// TIA Portal project "BatchSimulation_S71500" (V15)

(* hardware
DEVICE "S71500/ET200MP station_1"  S7-1500 station
   slot 0: "Rail_0"  Rack  6ES7 590-1***0-0AA0
   slot 1: "PLC_2_BatchController"  CPU 1512C-1 PN  6ES7 512-1CK01-0AB0  V2.5
      slot 3: "CPU display_1"  6ES7591-1AA00-0AA0
DEVICE "S71500/ET200MP station_2"  S7-1500 station
   slot 0: "Rail_0"  Rack  6ES7 590-1***0-0AA0
   slot 1: "PLC_1_Master"  CPU 1512C-1 PN  6ES7 512-1CK01-0AB0  V2.5
      slot 3: "CPU display_1"  6ES7591-1AA00-0AA0
*)

// ===== PLC "PLC_2_BatchController"  CPU 1512C-1 PN =====

VAR_GLOBAL   // PLC tag table "Default tag table"
   "Enable" AT %M100.0 : Bool;
   "Start" AT %M100.1 : Bool;
   "Estop" AT %M100.2 : Bool;
   "Ready" AT %M100.3 : Bool;
   "Setpoint" AT %MD150 : Real;
   "Vout" AT %MD154 : Real;
   "Running" AT %M100.4 : Bool;
   "State" AT %MW200 : Int;
   "Tag_1" AT %MD1000 : Real;
   "Tag_2" AT %MD1004 : DWord;
   "Tag_3" AT %M50.0 : Bool;
   "Tag_4" AT %M200.0 : Bool;
   "Tag_5" AT %MW204 : Int;
   "Tag_6" AT %M700.0 : Bool;
   "Tag_7" AT %MD200 : Real;
   "Tag_8" AT %MD300 : Real;
   "Tag_9" AT %M11.0 : Bool;
   "Tag_10" AT %M10.0 : Bool;
   "System_Byte" AT %MB1 : Byte;
   "FirstScan" AT %M1.0 : Bool;
   "DiagStatusUpdate" AT %M1.1 : Bool;
   "AlwaysTRUE" AT %M1.2 : Bool;
   "AlwaysFALSE" AT %M1.3 : Bool;
END_VAR

DATA_BLOCK "Batch1_Send"   // DB4
{ S7_Optimized_Access := 'FALSE' }
VERSION : 0.1
   VAR
      Ready : Bool;
      Running : Bool;
      Clock : Bool;
      Pulse : Int := 13;
      Vout : Real;
      ctrvalue : Real;
   END_VAR
BEGIN
END_DATA_BLOCK

DATA_BLOCK "Batch1_Recv"   // DB5
{ S7_Optimized_Access := 'FALSE' }
VERSION : 0.1
   VAR
      Start : Bool;
      Estop : Bool;
      Enable : Bool;
      PS : Int;
      Setpoint : Real;
   END_VAR
BEGIN
END_DATA_BLOCK

// folder: System blocks/Program resources

DATA_BLOCK "IEC_Timer_0_DB"   // DB1
{ S7_Optimized_Access := 'TRUE' }
AUTHOR : Simatic
FAMILY : IEC
NAME : IEC_TMR
VERSION : 1.0
// stored: InstanceOfName IEC_TIMER
"IEC_TIMER"
BEGIN
END_DATA_BLOCK

DATA_BLOCK "IEC_Timer_0_DB_1"   // DB2
{ S7_Optimized_Access := 'TRUE' }
AUTHOR : Simatic
FAMILY : IEC
NAME : IEC_TMR
VERSION : 1.0
// stored: InstanceOfName IEC_TIMER
"IEC_TIMER"
BEGIN
END_DATA_BLOCK

// folder: (top level)

FUNCTION "ClockGenerator" : Void   // FC1, LAD
{ S7_Optimized_Access := 'TRUE' }
VERSION : 0.1
   VAR_INPUT
      "Flow (m3/h)" : Real;
      PS : Int;
   END_VAR
   VAR_IN_OUT
      clock : Bool;
   END_VAR
   VAR_TEMP
      timing_ms : Int;
      timing : Time;
   END_VAR
BEGIN

REGION Network 1
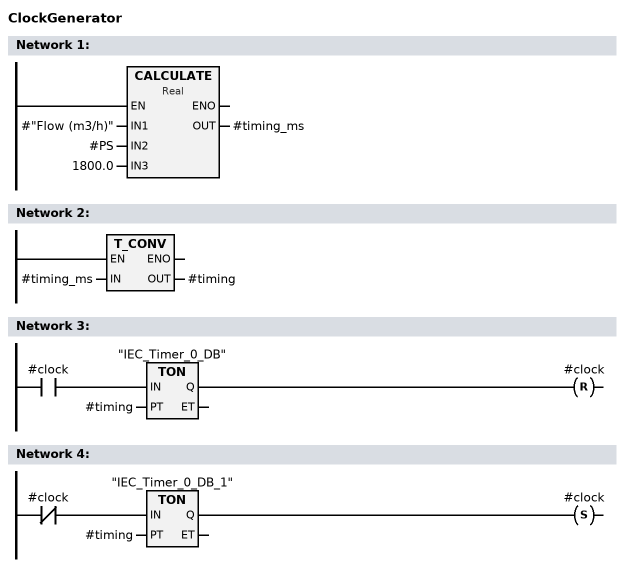
   RUNG wire#powerrail
      { S7_Templates := "SrcType := Real"; S7_Expression := "IN3/(IN1*IN2)" } Calculate(in1 := #"Flow (m3/h)", in2 := #PS, in3 := 1800.0, out => #timing_ms)
   END_RUNG
   // the same network as SCL:
   #timing_ms := 1800.0/(#"Flow (m3/h)"*#PS);
END_REGION

REGION Network 2
   #timing := T_CONV(IN := #timing_ms);
END_REGION

REGION Network 3
   "IEC_Timer_0_DB".TON(IN := #clock, PT := #timing);
   IF "IEC_Timer_0_DB".Q THEN #clock := FALSE; END_IF;
END_REGION

REGION Network 4
   "IEC_Timer_0_DB_1".TON(IN := NOT #clock, PT := #timing);
   IF "IEC_Timer_0_DB_1".Q THEN #clock := TRUE; END_IF;
END_REGION
END_FUNCTION

FUNCTION "BatchSimulation" : Void   // FC2, LAD
{ S7_Optimized_Access := 'TRUE' }
VERSION : 0.1
   VAR_INPUT
      Enable : Bool;
      Start : Bool;
      Estop : Bool;
      Setpoint : Real;
      PS : Int;
   END_VAR
   VAR_OUTPUT
      Ready : Bool;
   END_VAR
   VAR_IN_OUT
      "Vout(m3)" : Real;
      Running : Bool;
      pulse : Int;
      ctrlvalue : Real;
      clock : Bool;
   END_VAR
   VAR_TEMP
      flow : Real;
      tmp_clock : Bool;
      tmp_running : Bool;
   END_VAR
   VAR_TEMP   // added for the SCL form of the ladder/FBD networks
      _w1 : Bool;
   END_VAR
BEGIN

REGION Network 1: logic control
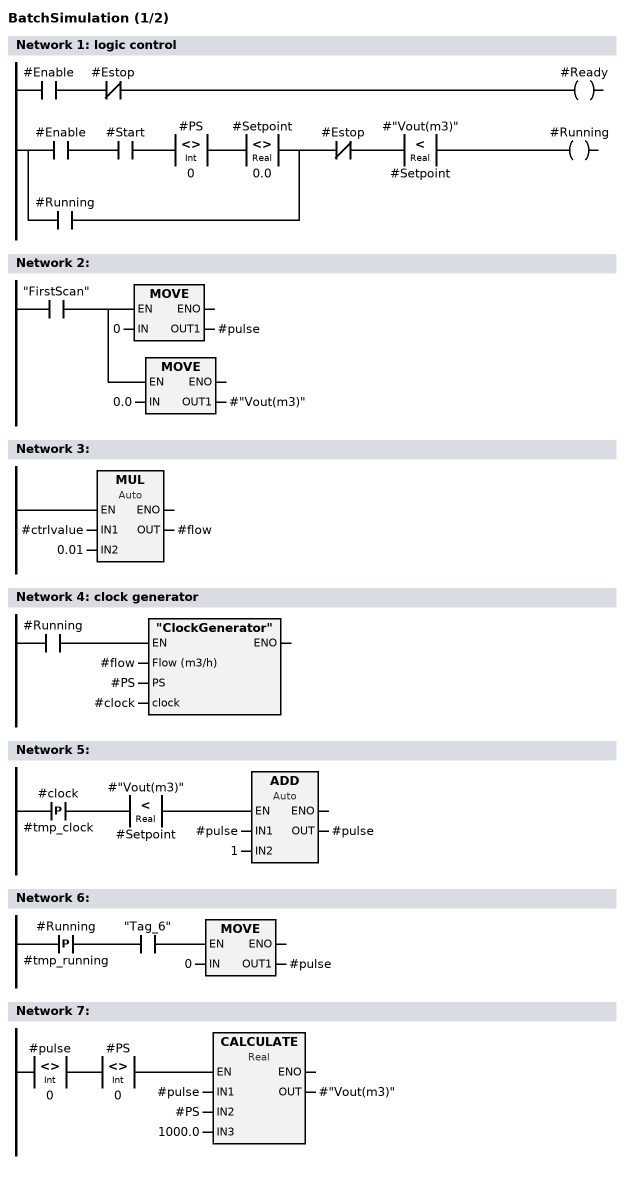
   RUNG wire#powerrail
      Contact( #Enable )
      I_Contact( #Estop )
      Coil( #Ready )
   END_RUNG
   RUNG wire#powerrail
      Contact( #Enable )
      Contact( #Start )
      { S7_Templates := "SrcType := Int" } NE_Contact(in1 := #PS, in2 := 0)
      { S7_Templates := "SrcType := Real" } NE_Contact(in1 := #Setpoint, in2 := 0.0)
      wire#w1
      I_Contact( #Estop )
      { S7_Templates := "SrcType := Real" } LT_Contact(in1 := #"Vout(m3)", in2 := #Setpoint)
      Coil( #Running )
   END_RUNG
   RUNG wire#powerrail
      Contact( #Running )
   END_RUNG wire#w1
   // the same network as SCL:
   #Ready := #Enable AND NOT #Estop;
   #Running := ((#Enable AND #Start AND (#PS <> 0) AND (#Setpoint <> 0.0)) OR #Running) AND NOT #Estop AND (#"Vout(m3)" < #Setpoint);
END_REGION

REGION Network 2
   RUNG wire#powerrail
      Contact( "FirstScan" )
      wire#w1
      Move(in := 0, out1 => #pulse)
   END_RUNG
   RUNG wire#w1
      Move(in := 0.0, out1 => #"Vout(m3)")
   END_RUNG
   // the same network as SCL:
   IF "FirstScan" THEN
       #pulse := 0;
       #"Vout(m3)" := 0.0;
   END_IF;
END_REGION

REGION Network 3
   RUNG wire#powerrail
      Mul(in1 := #ctrlvalue, in2 := 0.01, out => #flow)
   END_RUNG
   // the same network as SCL:
   #flow := #ctrlvalue * 0.01;
END_REGION

REGION Network 4: clock generator
   RUNG wire#powerrail
      Contact( #Running )
      "ClockGenerator"("Flow (m3/h)" := #flow, PS := #PS, clock := #clock)
   END_RUNG
   // the same network as SCL:
   IF #Running THEN "ClockGenerator"("Flow (m3/h)" := #flow, PS := #PS, clock := #clock); END_IF;
END_REGION

REGION Network 5
   RUNG wire#powerrail
      P_Contact(operand := #clock, bit := #tmp_clock)
      { S7_Templates := "SrcType := Real" } LT_Contact(in1 := #"Vout(m3)", in2 := #Setpoint)
      Add(in1 := #pulse, in2 := 1, out => #pulse)
   END_RUNG
   // the same network as SCL:
   #_w1 := #clock AND NOT #tmp_clock;   // rising edge of #clock
   #tmp_clock := #clock;
   IF #_w1 AND (#"Vout(m3)" < #Setpoint) THEN #pulse := #pulse + 1; END_IF;
END_REGION

REGION Network 6
   RUNG wire#powerrail
      P_Contact(operand := #Running, bit := #tmp_running)
      Contact( "Tag_6" )
      Move(in := 0, out1 => #pulse)
   END_RUNG
   // the same network as SCL:
   #_w1 := #Running AND NOT #tmp_running;   // rising edge of #Running
   #tmp_running := #Running;
   IF #_w1 AND "Tag_6" THEN #pulse := 0; END_IF;
END_REGION

REGION Network 7
   RUNG wire#powerrail
      { S7_Templates := "SrcType := Int" } NE_Contact(in1 := #pulse, in2 := 0)
      { S7_Templates := "SrcType := Int" } NE_Contact(in1 := #PS, in2 := 0)
      { S7_Templates := "SrcType := Real"; S7_Expression := "(IN1/IN2)/IN3" } Calculate(in1 := #pulse, in2 := #PS, in3 := 1000.0, out => #"Vout(m3)")
   END_RUNG
   // the same network as SCL:
   IF (#pulse <> 0) AND (#PS <> 0) THEN #"Vout(m3)" := (#pulse/#PS)/1000.0; END_IF;
END_REGION

REGION Network 8
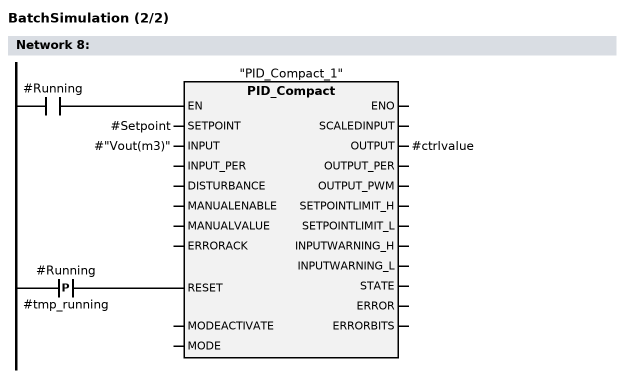
   #_w1 := #Running AND NOT #tmp_running;   // rising edge of #Running
   #tmp_running := #Running;
   IF #Running THEN
       "PID_Compact_1"(Setpoint := #Setpoint, Input := #"Vout(m3)", Reset := #_w1, Output => #ctrlvalue);   // PID_Compact
   END_IF;
END_REGION
END_FUNCTION

ORGANIZATION_BLOCK "Main"   // OB1, LAD, ProgramCycle
TITLE = "Main Program Sweep (Cycle)"
{ S7_Optimized_Access := 'TRUE' }
VERSION : 0.1
   VAR_INPUT
      Initial_Call : Bool;   // Initial call of this OB
      Remanence : Bool;   // =True, if remanent data are available
   END_VAR
BEGIN

REGION Network 1
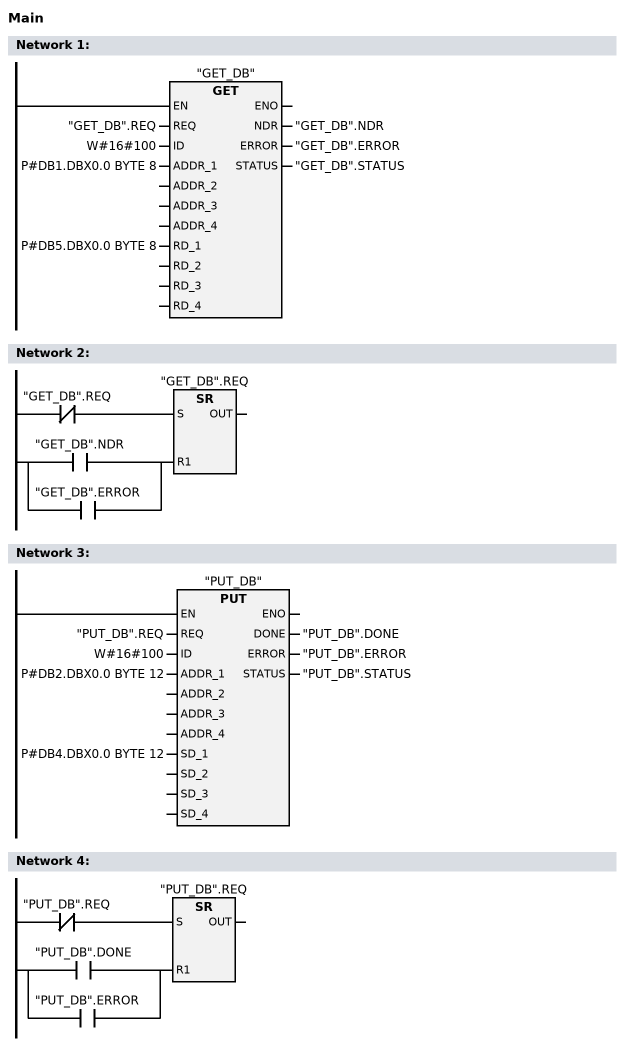
   "GET_DB"(REQ := "GET_DB".REQ,   // GET
            ID := W#16#100,
            ADDR_1 := P#DB1.DBX0.0 BYTE 8,
            RD_1 := P#DB5.DBX0.0 BYTE 8,
            NDR => "GET_DB".NDR,
            ERROR => "GET_DB".ERROR,
            STATUS => "GET_DB".STATUS);
END_REGION

REGION Network 2
   RUNG wire#powerrail
      I_Contact( "GET_DB".REQ )
      S_SR(operand := "GET_DB".REQ, r1 := wire#w1)
   END_RUNG
   RUNG wire#powerrail
      Contact( "GET_DB".NDR )
   END_RUNG wire#w1
   RUNG wire#powerrail
      Contact( "GET_DB".ERROR )
   END_RUNG wire#w1
   // the same network as SCL:
   IF NOT "GET_DB".REQ THEN
       "GET_DB".REQ := TRUE;   // SR flip-flop
   END_IF;
   IF "GET_DB".NDR OR "GET_DB".ERROR THEN "GET_DB".REQ := FALSE; END_IF;
END_REGION

REGION Network 3
   "PUT_DB"(REQ := "PUT_DB".REQ,   // PUT
            ID := W#16#100,
            ADDR_1 := P#DB2.DBX0.0 BYTE 12,
            SD_1 := P#DB4.DBX0.0 BYTE 12,
            DONE => "PUT_DB".DONE,
            ERROR => "PUT_DB".ERROR,
            STATUS => "PUT_DB".STATUS);
END_REGION

REGION Network 4
   RUNG wire#powerrail
      I_Contact( "PUT_DB".REQ )
      S_SR(operand := "PUT_DB".REQ, r1 := wire#w1)
   END_RUNG
   RUNG wire#powerrail
      Contact( "PUT_DB".DONE )
   END_RUNG wire#w1
   RUNG wire#powerrail
      Contact( "PUT_DB".ERROR )
   END_RUNG wire#w1
   // the same network as SCL:
   IF NOT "PUT_DB".REQ THEN
       "PUT_DB".REQ := TRUE;   // SR flip-flop
   END_IF;
   IF "PUT_DB".DONE OR "PUT_DB".ERROR THEN "PUT_DB".REQ := FALSE; END_IF;
END_REGION
END_ORGANIZATION_BLOCK

ORGANIZATION_BLOCK "Cyclic interrupt"   // OB30, LAD, CyclicInterrupt
{ S7_Optimized_Access := 'TRUE' }
VERSION : 0.1
   VAR_INPUT
      Initial_Call : Bool;   // Initial call of this OB
      Event_Count : Int;   // Events discarded
   END_VAR
BEGIN

REGION Network 1
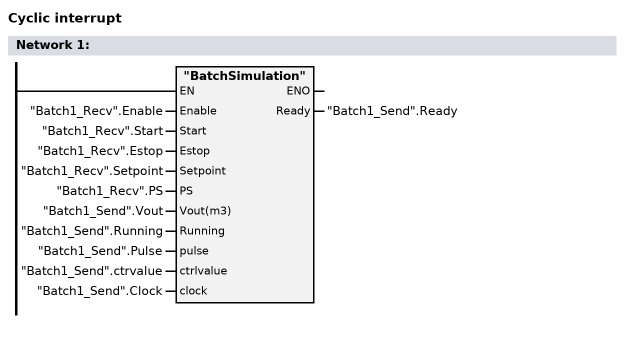
   RUNG wire#powerrail
      "BatchSimulation"(Enable := "Batch1_Recv".Enable, Start := "Batch1_Recv".Start, Estop := "Batch1_Recv".Estop, Setpoint := "Batch1_Recv".Setpoint, PS := "Batch1_Recv".PS, "Vout(m3)" := "Batch1_Send".Vout, Running := "Batch1_Send".Running, pulse := "Batch1_Send".Pulse, ctrlvalue := "Batch1_Send".ctrvalue, clock := "Batch1_Send".Clock, Ready => "Batch1_Send".Ready)
   END_RUNG
   // the same network as SCL:
   "BatchSimulation"(Enable := "Batch1_Recv".Enable,
                     Start := "Batch1_Recv".Start,
                     Estop := "Batch1_Recv".Estop,
                     Setpoint := "Batch1_Recv".Setpoint,
                     PS := "Batch1_Recv".PS,
                     "Vout(m3)" := "Batch1_Send".Vout,
                     Running := "Batch1_Send".Running,
                     pulse := "Batch1_Send".Pulse,
                     ctrlvalue := "Batch1_Send".ctrvalue,
                     clock := "Batch1_Send".Clock,
                     Ready => "Batch1_Send".Ready);
END_REGION
END_ORGANIZATION_BLOCK

// ===== PLC "PLC_1_Master"  CPU 1512C-1 PN =====

DATA_BLOCK "Diezel1_Send"   // DB1
{ S7_Optimized_Access := 'FALSE' }
VERSION : 0.1
   VAR
      Start : Bool;
      Estop : Bool;
      Enable : Bool;
      PS : Int := 13;
      Setpoint : Real;
   END_VAR
BEGIN
END_DATA_BLOCK

DATA_BLOCK "Diezel1_Recv"   // DB2
{ S7_Optimized_Access := 'FALSE' }
VERSION : 0.1
   VAR
      Ready : Bool;
      Running : Bool;
      Clock : Bool;
      Pulse : Int := 13;
      Vout : Real;
      ctrvalue : Real;
   END_VAR
BEGIN
END_DATA_BLOCK

DATA_BLOCK "Diezel_Common"   // DB5
{ S7_Optimized_Access := 'TRUE' }
VERSION : 0.1
   VAR
      Temp : Real := 25.0;
      Level : Real := 10.0;
      InitialLevel : Real := 10.0;
      BaseArea : Real := 10.0;
      Volume : Real;
      InitialVolume : Real;
      Flow1 : Real;
      Flow2 : Real;
   END_VAR
BEGIN
END_DATA_BLOCK

DATA_BLOCK "Diezel2_Recv"   // DB6
{ S7_Optimized_Access := 'FALSE' }
VERSION : 0.1
   VAR
      Ready : Bool;
      Running : Bool;
      Clock : Bool;
      Pulse : Int := 13;
      Vout : Real;
      ctrvalue : Real;
   END_VAR
BEGIN
END_DATA_BLOCK

DATA_BLOCK "Diezel2_Send"   // DB7
{ S7_Optimized_Access := 'FALSE' }
VERSION : 0.1
   VAR
      Start : Bool;
      Estop : Bool;
      Enable : Bool;
      PS : Int := 13;
      Setpoint : Real;
   END_VAR
BEGIN
END_DATA_BLOCK

FUNCTION "DiezelProcess" : Void   // FC1, LAD
{ S7_Optimized_Access := 'TRUE' }
VERSION : 0.1
   VAR_INPUT
      SendBytes : Bool;
      RecvBytes : Bool;
   END_VAR
   VAR_IN_OUT
      DB_Master_Send : DB_ANY;
      DB_Master_Recv : DB_ANY;
      DB_Batch_Send : DB_ANY;
      DB_Batch_Recv : DB_ANY;
      MyDB : Variant;
   END_VAR
BEGIN

REGION Network 1
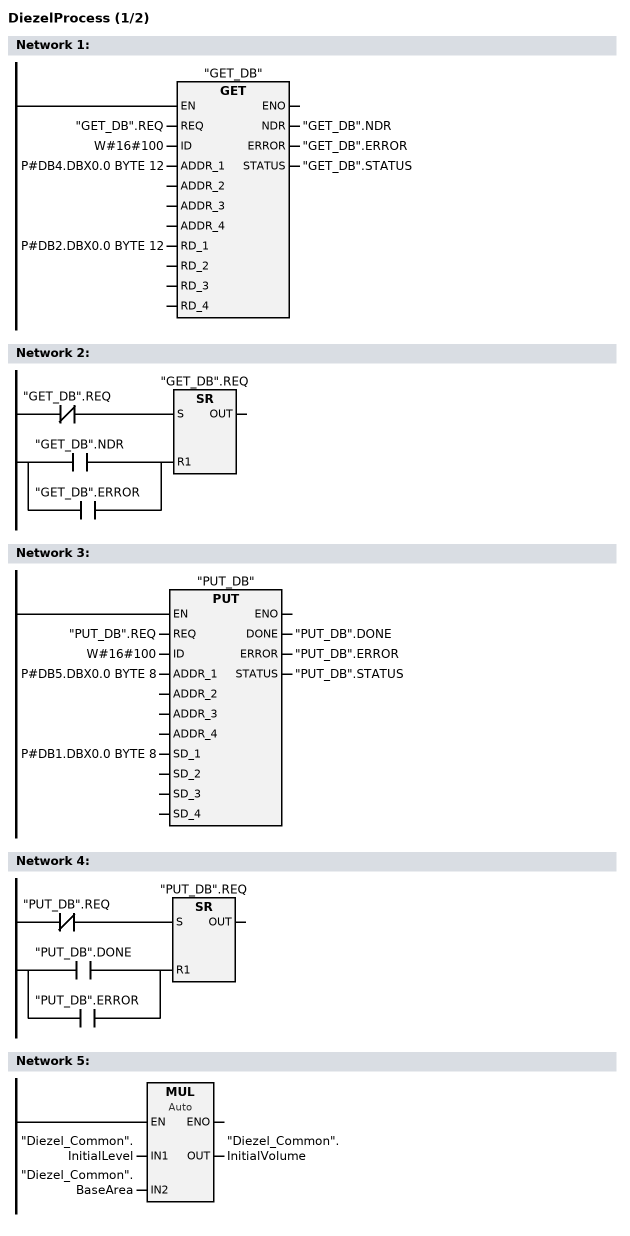
   "GET_DB"(REQ := "GET_DB".REQ,   // GET
            ID := W#16#100,
            ADDR_1 := P#DB4.DBX0.0 BYTE 12,
            RD_1 := P#DB2.DBX0.0 BYTE 12,
            NDR => "GET_DB".NDR,
            ERROR => "GET_DB".ERROR,
            STATUS => "GET_DB".STATUS);
END_REGION

REGION Network 2
   RUNG wire#powerrail
      I_Contact( "GET_DB".REQ )
      S_SR(operand := "GET_DB".REQ, r1 := wire#w1)
   END_RUNG
   RUNG wire#powerrail
      Contact( "GET_DB".NDR )
   END_RUNG wire#w1
   RUNG wire#powerrail
      Contact( "GET_DB".ERROR )
   END_RUNG wire#w1
   // the same network as SCL:
   IF NOT "GET_DB".REQ THEN
       "GET_DB".REQ := TRUE;   // SR flip-flop
   END_IF;
   IF "GET_DB".NDR OR "GET_DB".ERROR THEN "GET_DB".REQ := FALSE; END_IF;
END_REGION

REGION Network 3
   "PUT_DB"(REQ := "PUT_DB".REQ,   // PUT
            ID := W#16#100,
            ADDR_1 := P#DB5.DBX0.0 BYTE 8,
            SD_1 := P#DB1.DBX0.0 BYTE 8,
            DONE => "PUT_DB".DONE,
            ERROR => "PUT_DB".ERROR,
            STATUS => "PUT_DB".STATUS);
END_REGION

REGION Network 4
   RUNG wire#powerrail
      I_Contact( "PUT_DB".REQ )
      S_SR(operand := "PUT_DB".REQ, r1 := wire#w1)
   END_RUNG
   RUNG wire#powerrail
      Contact( "PUT_DB".DONE )
   END_RUNG wire#w1
   RUNG wire#powerrail
      Contact( "PUT_DB".ERROR )
   END_RUNG wire#w1
   // the same network as SCL:
   IF NOT "PUT_DB".REQ THEN
       "PUT_DB".REQ := TRUE;   // SR flip-flop
   END_IF;
   IF "PUT_DB".DONE OR "PUT_DB".ERROR THEN "PUT_DB".REQ := FALSE; END_IF;
END_REGION

REGION Network 5
   RUNG wire#powerrail
      Mul(in1 := "Diezel_Common".InitialLevel, in2 := "Diezel_Common".BaseArea, out => "Diezel_Common".InitialVolume)
   END_RUNG
   // the same network as SCL:
   "Diezel_Common".InitialVolume := "Diezel_Common".InitialLevel * "Diezel_Common".BaseArea;
END_REGION

REGION Network 6
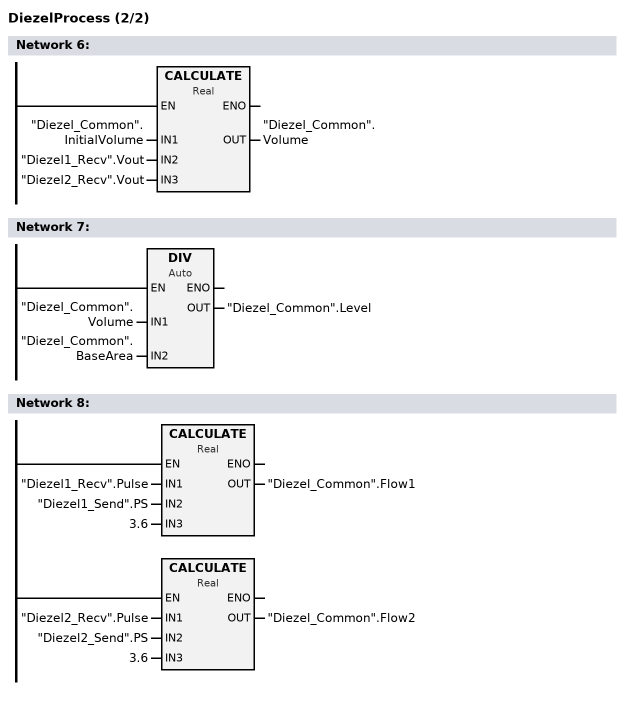
   RUNG wire#powerrail
      { S7_Templates := "SrcType := Real"; S7_Expression := "IN1-IN2-IN3" } Calculate(in1 := "Diezel_Common".InitialVolume, in2 := "Diezel1_Recv".Vout, in3 := "Diezel2_Recv".Vout, out => "Diezel_Common".Volume)
   END_RUNG
   // the same network as SCL:
   "Diezel_Common".Volume := "Diezel_Common".InitialVolume-"Diezel1_Recv".Vout-"Diezel2_Recv".Vout;
END_REGION

REGION Network 7
   RUNG wire#powerrail
      Div(in1 := "Diezel_Common".Volume, in2 := "Diezel_Common".BaseArea, out => "Diezel_Common".Level)
   END_RUNG
   // the same network as SCL:
   "Diezel_Common".Level := "Diezel_Common".Volume / "Diezel_Common".BaseArea;
END_REGION

REGION Network 8
   RUNG wire#powerrail
      { S7_Templates := "SrcType := Real"; S7_Expression := "IN1*IN2/IN3" } Calculate(in1 := "Diezel1_Recv".Pulse, in2 := "Diezel1_Send".PS, in3 := 3.6, out => "Diezel_Common".Flow1)
   END_RUNG
   RUNG wire#powerrail
      { S7_Templates := "SrcType := Real"; S7_Expression := "IN1*IN2/IN3" } Calculate(in1 := "Diezel2_Recv".Pulse, in2 := "Diezel2_Send".PS, in3 := 3.6, out => "Diezel_Common".Flow2)
   END_RUNG
   // the same network as SCL:
   "Diezel_Common".Flow1 := "Diezel1_Recv".Pulse*"Diezel1_Send".PS/3.6;
   "Diezel_Common".Flow2 := "Diezel2_Recv".Pulse*"Diezel2_Send".PS/3.6;
END_REGION
END_FUNCTION

ORGANIZATION_BLOCK "Main"   // OB1, LAD, ProgramCycle
TITLE = "Main Program Sweep (Cycle)"
{ S7_Optimized_Access := 'TRUE' }
VERSION : 0.1
   VAR_INPUT
      Initial_Call : Bool;   // Initial call of this OB
      Remanence : Bool;   // =True, if remanent data are available
   END_VAR
BEGIN

REGION Network 1
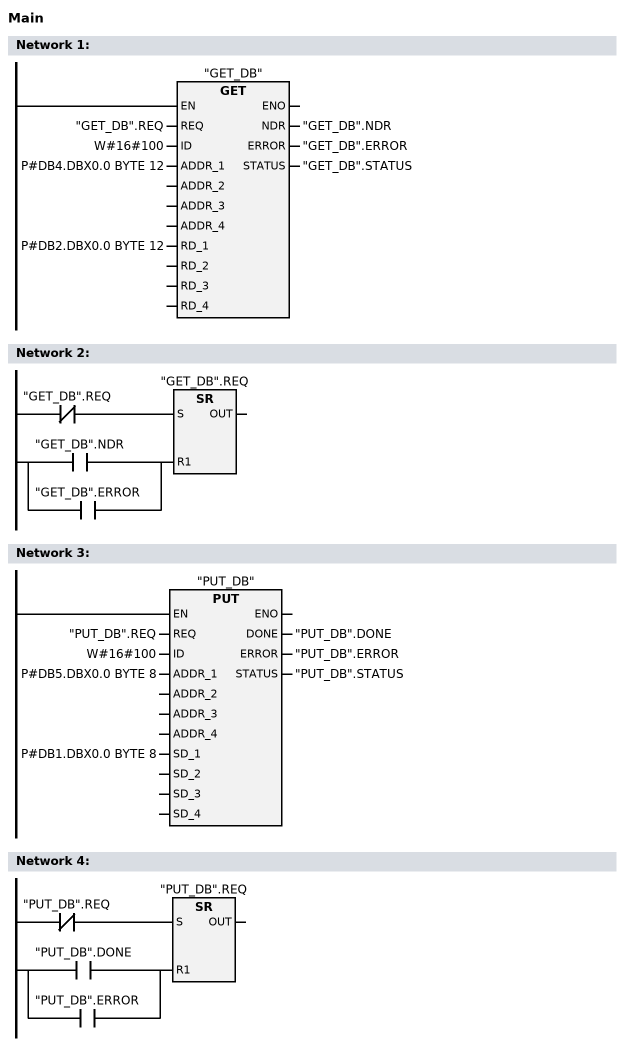
   "GET_DB"(REQ := "GET_DB".REQ,   // GET
            ID := W#16#100,
            ADDR_1 := P#DB4.DBX0.0 BYTE 12,
            RD_1 := P#DB2.DBX0.0 BYTE 12,
            NDR => "GET_DB".NDR,
            ERROR => "GET_DB".ERROR,
            STATUS => "GET_DB".STATUS);
END_REGION

REGION Network 2
   RUNG wire#powerrail
      I_Contact( "GET_DB".REQ )
      S_SR(operand := "GET_DB".REQ, r1 := wire#w1)
   END_RUNG
   RUNG wire#powerrail
      Contact( "GET_DB".NDR )
   END_RUNG wire#w1
   RUNG wire#powerrail
      Contact( "GET_DB".ERROR )
   END_RUNG wire#w1
   // the same network as SCL:
   IF NOT "GET_DB".REQ THEN
       "GET_DB".REQ := TRUE;   // SR flip-flop
   END_IF;
   IF "GET_DB".NDR OR "GET_DB".ERROR THEN "GET_DB".REQ := FALSE; END_IF;
END_REGION

REGION Network 3
   "PUT_DB"(REQ := "PUT_DB".REQ,   // PUT
            ID := W#16#100,
            ADDR_1 := P#DB5.DBX0.0 BYTE 8,
            SD_1 := P#DB1.DBX0.0 BYTE 8,
            DONE => "PUT_DB".DONE,
            ERROR => "PUT_DB".ERROR,
            STATUS => "PUT_DB".STATUS);
END_REGION

REGION Network 4
   RUNG wire#powerrail
      I_Contact( "PUT_DB".REQ )
      S_SR(operand := "PUT_DB".REQ, r1 := wire#w1)
   END_RUNG
   RUNG wire#powerrail
      Contact( "PUT_DB".DONE )
   END_RUNG wire#w1
   RUNG wire#powerrail
      Contact( "PUT_DB".ERROR )
   END_RUNG wire#w1
   // the same network as SCL:
   IF NOT "PUT_DB".REQ THEN
       "PUT_DB".REQ := TRUE;   // SR flip-flop
   END_IF;
   IF "PUT_DB".DONE OR "PUT_DB".ERROR THEN "PUT_DB".REQ := FALSE; END_IF;
END_REGION
END_ORGANIZATION_BLOCK